Universal Robots PolyScope program: Wheel_holder.urp

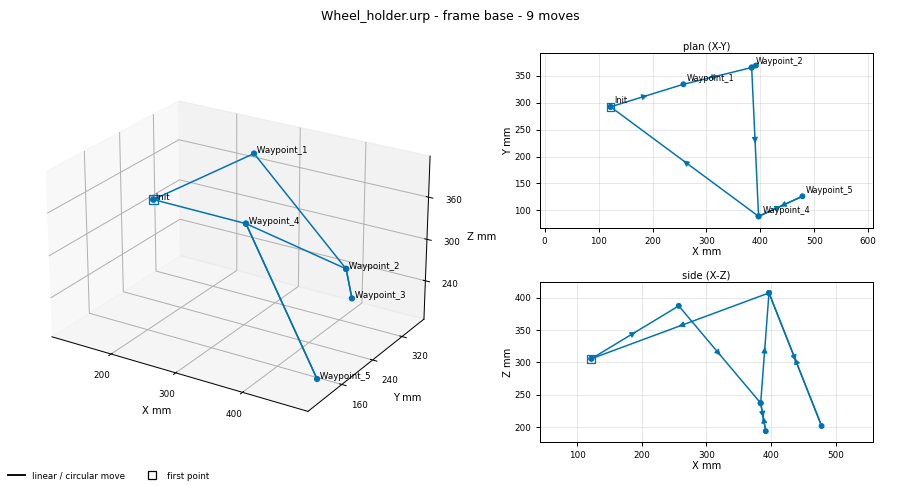
[picture p0: tool path of Wheel_holder.urp in frame base, 9 of 9 moves have a stored position in this frame; points joined in program order, loops and branches not executed]
Program Wheel_holder (installation=default directory=/programs/Mursal createdIn=5.11.11.1010533 lastSavedIn=5.11.11.1010533 robotSerialNumber=20205300864)
Calibrated DH parameters: a=[-0.000166, -0.243494, -0.153108, 0.000057, -0.000123, 0]; d=[0.151897, -1.34267, 53.988124, -52.514559, 0.085283, 0.092193]; alpha=[1.572472, -0.003756, 0.002824, 1.570807, -1.572621, 0]; deltaTheta=[0, 0.020704, 7.033215, -0.770746, 0.000004, 0]
Robot Program (runOnlyOnce=true)
  MoveL speed 250 mm/s, acceleration 1200 mm/s^2 (useActiveTCP=true) feature=Base
    Waypoint Init: TCP in base x=122.11 y=292.123 z=305.739 mm, rx=1.1347 ry=-2.9295 rz=-0.0001 rad; joints [91.642, -87.587, -91.765, -90.542, 90.033, 859.397] deg
    Waypoint Waypoint_1: TCP in base x=257.155 y=333.945 z=387.357 mm, rx=0.3044 ry=-3.1042 rz=-0.0213 rad; joints [70.261, -138.666, 10.13, -141.202, 91.226, 869.047] deg
    Waypoint Waypoint_2: TCP in base x=383.738 y=364.987 z=237.054 mm, rx=-0.0826 ry=3.109 rz=0.0851 rad; joints [57.863, -155.006, -6.065, -105.252, 90.075, 864.767] deg
    Waypoint Waypoint_3: TCP in base x=391.63 y=368.708 z=193.676 mm, rx=0.0866 ry=-3.1404 rz=0 rad; joints [57.396, -161.638, -2.721, -105.537, 89.783, 864.171] deg
    URCap Gripper (Robotiq_Grippers, Robotiq Inc.) dataModel(position=80.3921568627451, force=0.0, speed=100.0, positionInDouble=80.3921568627451, forceInDouble=0.0, speedInDouble=100.0, slaveIds=[9], blocking=true, robotCompliant=false)
    Waypoint Waypoint_2: TCP in base x=383.738 y=364.987 z=237.054 mm, rx=-0.0826 ry=3.109 rz=0.0851 rad; joints [57.863, -155.006, -6.065, -105.252, 90.075, 864.767] deg
    Waypoint Waypoint_4: TCP in base x=396.57 y=89.083 z=407.361 mm, rx=-0.1467 ry=3.0438 rz=0.051 rad; joints [31.826, -142.019, 24.603, -146.848, 88.756, 836.211] deg
    Waypoint Waypoint_5: TCP in base x=477.915 y=126.341 z=201.666 mm, rx=-0.0289 ry=-3.1414 rz=0.0001 rad; joints [30.118, -137.429, -48.681, -83.79, 89.877, 841.221] deg
    URCap Gripper (Robotiq_Grippers, Robotiq Inc.) dataModel(position=0.0, force=0.0, speed=100.0, positionInDouble=0.0, forceInDouble=0.0, speedInDouble=100.0, slaveIds=[9], blocking=true, robotCompliant=false)
    Waypoint Waypoint_4: TCP in base x=396.57 y=89.083 z=407.361 mm, rx=-0.1467 ry=3.0438 rz=0.051 rad; joints [31.826, -142.019, 24.603, -146.848, 88.756, 836.211] deg
    Waypoint Init: TCP in base x=122.11 y=292.123 z=305.739 mm, rx=1.1347 ry=-2.9295 rz=-0.0001 rad; joints [91.642, -87.587, -91.765, -90.542, 90.033, 859.397] deg
